Universal Robots PolyScope program: joang_p1.urp

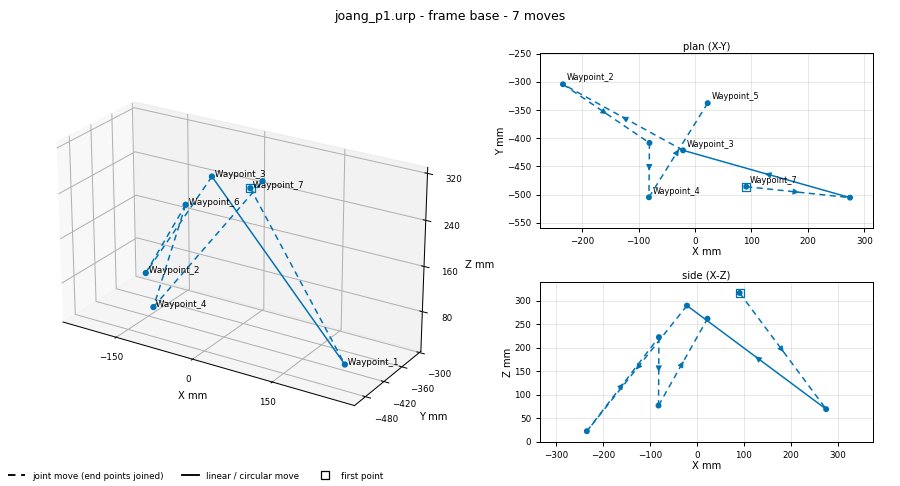
[picture p0: tool path of joang_p1.urp in frame base, 7 of 7 moves have a stored position in this frame; points joined in program order, loops and branches not executed]
Program joang_p1 (installation=default directory=/programs createdIn=5.14.5 lastSavedIn=5.14.5 robotSerialNumber=20195300809)
Calibrated DH parameters: a=[-0.000085, -0.20076, -0.212369, 0.000121, -0.000118, 0]; d=[0.15185, -26.306375, 24.753047, 1.684739, 0.085386, 0.092088]; alpha=[1.572149, -0.00522, -0.011864, 1.571339, -1.571085, 0]; deltaTheta=[0, 0.599885, -0.513355, -0.086555, 0.000006, 0]
InitVariablesNode
BeforeStart
  URCap Gripper Activate (Robotiq_Grippers, Robotiq Inc.) dataModel(ResetAndActivateKey=false)
  Script: socket_open("10.5.20.90",29999)
  Script: socket_send_string("hello pc")
Robot Program (runOnlyOnce=false)
  MoveJ speed 60 deg/s, acceleration 80 deg/s^2 (useActiveTCP=true) feature=Base
    Waypoint Waypoint_7: TCP in base x=90.834 y=-485.852 z=316.412 mm, rx=0.0237 ry=2.9457 rz=-0.7349 rad; joints [-59.15, -115.709, -22.923, -104.113, 80.211, 30.09] deg; TCP offset x=0 y=0 z=174 mm, rx=0 ry=0 rz=0 rad
  MoveJ speed 60 deg/s, acceleration 80 deg/s^2 (useActiveTCP=true) feature=Base
    Waypoint Waypoint_1: TCP in base x=274.791 y=-505.274 z=69.289 mm, rx=-0.0548 ry=2.9486 rz=-0.2932 rad; joints [-48.642, -143.201, -34.694, -76.846, 89.543, 39.453] deg
    URCap Gripper (Robotiq_Grippers, Robotiq Inc.) dataModel(position=58.8235294117647, force=0.0, speed=0.0, positionInDouble=58.8235294117647, forceInDouble=0.0, speedInDouble=0.0, slaveIds=[9], blocking=true)
    MoveL speed 250 mm/s, acceleration 1200 mm/s^2 (useActiveTCP=true) feature=Base
      Waypoint Waypoint_3: TCP in base x=-21.203 y=-421.42 z=289.45 mm, rx=-0.093 ry=-3.0455 rz=0.3937 rad; joints [-68.744, -113.884, -19.43, -124.693, 80.041, 24.518] deg
    MoveJ speed 60 deg/s, acceleration 80 deg/s^2 (useActiveTCP=true) feature=Base
      Waypoint Waypoint_2: TCP in base x=-234.099 y=-304.274 z=22.417 mm, rx=-0.017 ry=3.124 rz=-0.023 rad; joints [-108.673, -109.96, -95.435, -64.112, 90.581, -19.215] deg
      URCap Gripper (Robotiq_Grippers, Robotiq Inc.) dataModel(position=10.588235294117647, force=0.0, speed=0.0, positionInDouble=10.588235294117647, forceInDouble=0.0, speedInDouble=0.0, slaveIds=[9], blocking=true)
      URCap Gripper (Robotiq_Grippers, Robotiq Inc.) dataModel(position=56.07843137254902, force=0.0, speed=0.0, positionInDouble=56.07843137254902, forceInDouble=0.0, speedInDouble=0.0, slaveIds=[9], blocking=true)
    Set DigitalOutput pin=digital_out[0]; digitalValue=1
    MoveJ speed 60 deg/s, acceleration 80 deg/s^2 (useActiveTCP=true) feature=Base
      Waypoint Waypoint_6: TCP in base x=-80.793 y=-408.26 z=222.448 mm, rx=0.0639 ry=3.0417 rz=-0.5242 rad; joints [-83.307, -94.149, -72.111, -83.928, 89.709, 9.456] deg
    MoveJ speed 60 deg/s, acceleration 80 deg/s^2 (useActiveTCP=true) feature=Base
      Waypoint Waypoint_4: TCP in base x=-81.678 y=-504.668 z=76.906 mm, rx=-0.0639 ry=3.1163 rz=-0.1664 rad; joints [-84.918, -133.718, -44.594, -85.489, 89.902, 3.091] deg
      URCap Gripper (Robotiq_Grippers, Robotiq Inc.) dataModel(position=19.215686274509803, force=0.0, speed=0.0, positionInDouble=19.215686274509803, forceInDouble=0.0, speedInDouble=0.0, slaveIds=[9], blocking=true)
    MoveJ speed 60 deg/s, acceleration 80 deg/s^2 (useActiveTCP=true) feature=Base
      Waypoint Waypoint_5: TCP in base x=22.492 y=-337.762 z=261.698 mm, rx=-0.0816 ry=3.1105 rz=-0.0454 rad; joints [-64.512, -102.605, -37.785, -127.361, 90.397, 23.269] deg
      URCap Gripper (Robotiq_Grippers, Robotiq Inc.) dataModel(position=10.980392156862745, force=0.0, speed=0.0, positionInDouble=10.980392156862745, forceInDouble=0.0, speedInDouble=0.0, slaveIds=[9], blocking=true)
